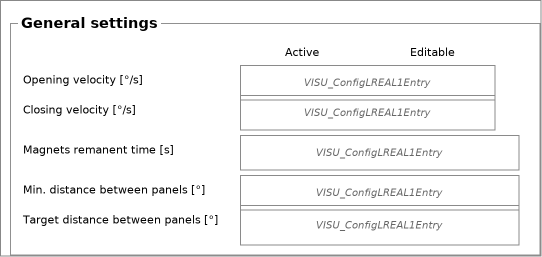
VISUALIZATION VISU_CoverConfig_General  // 542x257
VAR_IN_OUT
	activeConfig : CoverConfig;
    editableConfig : CoverConfig;
END_VAR
    GroupBox (10,15 530x240), "General settings"
        Label (10,50 175x30), "Opening velocity [°/s]"
        Label (10,80 175x30), "Closing velocity [°/s]"
        Label (10,160 190x30), "Min. distance between panels [°]"
        Label (360,25 125x25), "Editable"
        Label (230,25 125x25), "Active"
        Label (10,120 175x30), "Magnets remanent time [s]"
        Label (10,190 205x30), "Target distance between panels [°]"
        Frame (230,160 279x35)
            shows VISU_ConfigLREAL1Entry(active := activeConfig.minDistanceBetweenPanelSets, editable := editableConfig.minDistanceBetweenPanelSets)
        Frame (230,190 279x40)
            shows VISU_ConfigLREAL1Entry(active := activeConfig.targetDistanceBetweenPanelSets, editable := editableConfig.targetDistanceBetweenPanelSets)
        Frame (230,120 279x35)
            shows VISU_ConfigLREAL1Entry(active := activeConfig.magnetRemanentTime, editable := editableConfig.magnetRemanentTime)
        Frame (230,50 255x35)
            shows VISU_ConfigLREAL1Entry(active := activeConfig.openingVelocity, editable := editableConfig.openingVelocity)
        Frame (230,80 255x35)
            shows VISU_ConfigLREAL1Entry(active := activeConfig.closingVelocity, editable := editableConfig.closingVelocity)
END_VISUALIZATION

(* stored: Version 1.1.0.1, ProductVersion 3.1.4019.2
   Visu VISU_CoverConfig_General: Id {bae08b8a-6bb1-4cc7-b228-f234881dde6d} *)
